// TIA Portal V17 export
// export: Created 2025-01-08T13:55:34.1056765Z, ExportSetting WithDefaults, DisplayName Totally Integrated Automation Portal, DisplayVersion V17, DisplayName TIA Portal Openness, DisplayVersion V17, DisplayName TIA Portal Version Control Interface, DisplayVersion V17, DisplayName SINAMICS Startdrive Advanced, DisplayVersion V17 Update2, DisplayName SINAMICS Startdrive G130, G150, S120, S150, SINAMICS MV, S210, DisplayVersion V17 Update2, DisplayName SINAMICS Startdrive G110M, G120, G120C, G120D, G120P, G115D, DisplayVersion V17 Update2, DisplayName STEP 7 Professional, DisplayVersion V17, DisplayName STEP 7 Safety, DisplayVersion V17, DisplayName WinCC Advanced, DisplayVersion V17
DATA_BLOCK "DB - Btn_Tags"   // DB60
{ S7_Optimized_Access := 'FALSE' }
VERSION : 0.1
// stored: AutoNumber true, DBAccessibleFromOPCUA true, DBAccessibleFromWebserver true, IsOnlyStoredInLoadMemory false, IsWriteProtectedInAS false
   VAR RETAIN
      Starta_Banor : Bool;   // Starta Banor
      Reject_Topp_Pulse : Bool;   // Reject Topp
      Reject_Bottom_Pulse : Bool;   // Reject Botten
      Ignore_External_Pause : Bool;   // Ignorera External Pause
      MoveRotateProductCylinder : Bool;   // Rotera Dosa Cylinder
      Index_Wheel_Brake : Bool;   // Indexhjul Broms
      StandbyOff : Bool;   // Deaktivera Standby
      JogFunctionActive : Bool;   // Aktivera Jog
      Jog : Bool;   // Kör Jog
      Speed_1 : Bool;   // Hastighet 1
      Speed_2 : Bool;   // Hastighet 2
      Speed_3 : Bool;   // Hastighet 3
      EmptyMachine : Bool;   // Töm Maskin
      Activate_Cam1 : Bool;   // Aktivera Kamera 1
      Activate_Cam2 : Bool;   // Aktivera Kamera 2
      Activate_Cam3 : Bool;   // Aktivera Kamera 3
      Activate_Cam4 : Bool;   // Aktivera Kamera 4
      Speed_4 : Bool;   // Hastighet 4
      Speed_5 : Bool;   // Hastighet 5
      Disable_LabelAdjustMent : Bool;   // Deaktivera Etikettjustering
      Activate_Printer : Bool;   // Printer
   END_VAR
BEGIN
END_DATA_BLOCK
